(* CoDeSys 2.3 export: GENERATOR.EXP *)

(* POU EdgeDetector, ST *)
FUNCTION_BLOCK EdgeDetector
VAR_INPUT
	inputValue : BOOL;
END_VAR
VAR_OUTPUT
	risingEdge : BOOL;
	fallingEdge : BOOL;
END_VAR
VAR
	prev : BOOL := FALSE;
END_VAR
IF inputValue > prev THEN
	risingEdge := TRUE;
	fallingEdge := FALSE;
ELSIF inputValue < prev THEN
	risingEdge := FALSE;
	fallingEdge := TRUE;
ELSE
	risingEdge := FALSE;
	fallingEdge := FALSE;
END_IF
prev := inputValue;
END_FUNCTION_BLOCK

(* POU EdgeDetectorDouble, ST *)
FUNCTION_BLOCK EdgeDetectorDouble
VAR_INPUT
	inputValue : BOOL;
	threshold : INT;
END_VAR
VAR_OUTPUT
	risingEdge : BOOL;
	fallingEdge : BOOL;
	double : BOOL;
END_VAR
VAR
	prev : BOOL := FALSE;
	timer : INT := 0;
END_VAR
IF inputValue > prev THEN
	risingEdge := TRUE;
	fallingEdge := FALSE;
	IF timer < threshold THEN
		double := TRUE;
	ELSE
		double := FALSE;
	END_IF
	timer := 0;
ELSIF inputValue < prev THEN
	risingEdge := FALSE;
	fallingEdge := TRUE;
	IF timer < 32767 THEN
		timer := timer + 1;
	END_IF
	double := FALSE;
ELSE
	risingEdge := FALSE;
	fallingEdge := FALSE;
	IF timer < 32767 THEN
		timer := timer + 1;
	END_IF
	double := FALSE;
END_IF
prev := inputValue;
END_FUNCTION_BLOCK

(* POU PwmSignal, ST *)
FUNCTION PwmSignal : REAL
VAR_INPUT
	a : REAL;
	offset : REAL;
	w : REAL;
	t : INT;
	duty : REAL;
END_VAR
VAR
	per : INT;
END_VAR
per := REAL_TO_INT(F_TASK / w);
IF duty*per >= per THEN
	PwmSignal := offset + a;
ELSIF duty*per <=0 THEN
	PwmSignal := offset - a;
ELSIF (t MOD per) < duty*per THEN
	PwmSignal := offset + a;
ELSE
	PwmSignal := offset - a;
END_IF
END_FUNCTION

(* POU SinusFunction, ST *)
FUNCTION SinusFunction : REAL
VAR_INPUT
	a : REAL;
	offset : REAL;
	w : REAL;
	t : INT;
END_VAR
VAR
END_VAR
SinusFunction := a * SIN(INT_TO_REAL(t)*w /F_TASK *2.0*3.1415) + offset;
END_FUNCTION

(* POU SquareSignal, ST *)
FUNCTION SquareSignal : REAL
VAR_INPUT
	a : REAL;
	offset : REAL;
	w : REAL;
	t : INT;
END_VAR
VAR
	per : INT;
END_VAR
per := REAL_TO_INT(F_TASK / w);
IF (t MOD per) < (per / 2) THEN
	SquareSignal := offset + a;
ELSE
	SquareSignal := offset - a;
END_IF
END_FUNCTION
